INTERFACE I_WashStrategy

METHOD GetWashSettings 
VAR_INPUT
END_VAR
END_METHOD

METHOD ProgramName : BOOL
VAR_INPUT
	
END_VAR
END_METHOD

END_INTERFACE

(* stored: Version 1.1.0.1, ProductVersion 3.1.4024.16
   Itf I_WashStrategy: Id {ffeaff33-ef96-4576-8451-c0f0ea2434bd}
   Method GetWashSettings: Id {db05378f-6245-48d4-a5f4-9dfbf332898e}
   Method ProgramName: Id {d02b7e03-2a62-429f-bdf5-420156f9dc45} *)
